// TIA Portal project "Apple_Juice_Process_System" (V15)
// Vorlageprojekt für das Buch mit Zielsystem S7-1200

(* hardware
DEVICE "S7-1200-Station_1"  S7-1200 Station
   slot 0: "Baugruppenträger_0"  Rack  V1.0
   slot 1: "PLC_1"  CPU 1211C DC/DC/DC  6ES7 211-1AE40-0XB0  V4.1
*)

// ===== PLC "PLC_1"  CPU 1211C DC/DC/DC =====

VAR_GLOBAL   // PLC tag table "Standard-Variablentabelle"
   "Tag_1" AT %Q1.6 : Bool;
   "Tag_2" AT %I1.5 : Bool;
   "Tag_3" AT %I1.6 : Bool;
   "System_Byte" AT %MB1 : Byte;
   "FirstScan" AT %M1.0 : Bool;
   "DiagStatusUpdate" AT %M1.1 : Bool;
   "AlwaysTRUE" AT %M1.2 : Bool;
   "AlwaysFALSE" AT %M1.3 : Bool;
   "Clock_Byte" AT %MB0 : Byte;
   "Clock_10Hz" AT %M0.0 : Bool;
   "Clock_5Hz" AT %M0.1 : Bool;
   "Clock_2.5Hz" AT %M0.2 : Bool;
   "Clock_2Hz" AT %M0.3 : Bool;
   "Clock_1.25Hz" AT %M0.4 : Bool;
   "Clock_1Hz" AT %M0.5 : Bool;
   "Clock_0.625Hz" AT %M0.6 : Bool;
   "Clock_0.5Hz" AT %M0.7 : Bool;
END_VAR

VAR_GLOBAL   // PLC tag table "I/O"
   "EMERGENCY_BUTTON" AT %I0.0 : Bool;
   "START_BUTTON" AT %I0.1 : Bool;
   "STOP_BUTTON" AT %I0.2 : Bool;
   "WATER_FLOW_METER" AT %ID30 : DWord;
   "WATER_LEVEL_METER" AT %ID34 : DWord;
   "APPLE_JUICE_FLOW_METER" AT %ID38 : DWord;
   "APPLE_JUICE_LEVEL_METER" AT %ID42 : DWord;
   "APPLE_FLOW_METER" AT %ID46 : DWord;
   "APPLE_LEVEL_METER" AT %ID50 : DWord;
   "ROLLER_ENABLE_0" AT %Q0.7 : Bool;
   "START_BUTTON_LIGHT" AT %Q0.1 : Bool;
   "STOP_BUTTON_LIGHT" AT %Q0.2 : Bool;
   "RESET_BUTTON_LIGHT" AT %Q0.3 : Bool;
   "WATER_CHARGE_VALVE" AT %QD30 : DWord;
   "WATER_DISCHARGE_VALVE" AT %QD34 : DWord;
   "APPLE_JUICE_CHARGE_VALVE" AT %QD38 : DWord;
   "APPLE_JUICE_DISCHARGE_VALVE" AT %QD42 : DWord;
   "APPLE_CHARGE_VALVE" AT %QD46 : DWord;
   "APPLE_DISCHARGE_VALVE" AT %QD50 : DWord;
   "PRODUCTION_ENABLE" AT %I0.3 : Bool;
   "PRODUCTION_DISABLE" AT %I0.4 : Bool;
   "APPLE_JUICE_AMOUNT_SET" AT %ID54 : DWord;
   "GREEN_LIGHT" AT %Q0.4 : Bool;
   "YELLOW_LIGHT" AT %Q0.5 : Bool;
   "RED_LIGHT" AT %Q0.6 : Bool;
   "HMI" AT %QD54 : DWord;
   "BOTTLE_LEFT" AT %I0.5 : Bool;
   "RESET_BUTTON" AT %I0.6 : Bool;
   "ROLLER_ENABLE_1" AT %Q1.0 : Bool;
   "ROLLER_ENABLE_2" AT %Q1.1 : Bool;
   "ROLLER_ENABLE_3" AT %Q1.2 : Bool;
END_VAR

DATA_BLOCK "main_prog_DB"   // DB1
{ S7_Optimized_Access := 'TRUE' }
VERSION : 0.1
// stored: InstanceOfName main_prog
"main_prog"
BEGIN
END_DATA_BLOCK

// folder: System blocks/Program resources

DATA_BLOCK "IEC_Timer_0_DB"   // DB7
{ S7_Optimized_Access := 'TRUE' }
AUTHOR : Simatic
FAMILY : IEC
NAME : IEC_TMR
VERSION : 1.0
// stored: InstanceOfName IEC_TIMER
"IEC_TIMER"
BEGIN
END_DATA_BLOCK

// folder: (top level)

FUNCTION_BLOCK "main_prog"   // FB1, SCL
{ S7_Optimized_Access := 'TRUE' }
VERSION : 0.1
   VAR_INPUT
      emergencyButton : Bool;
      startButton : Bool;
      stopButton : Bool;
      resetButton : Bool;
      productionEnable : Bool;
      productionDisable : Bool;
      bottleLeft : Bool;
      waterFlowMeter : Real;
      waterLevelMeter : Real;
      appleJuiceFlowMeter : Real;
      appleJuiceLevelMeter : Real;
      appleFlowMeter : Real;
      appleLevelMeter : Real;
      appleJuiceAmountSet : Real;
   END_VAR
   VAR_OUTPUT
      rollerEnable0 : Bool;
      rollerEnable1 : Bool;
      rollerEnable2 : Bool;
      rollerEnable3 : Bool;
      startButtonLight : Bool;
      stopButtonLight : Bool;
      resetButtonLight : Bool;
      greenLight : Bool;
      yellowLight : Bool;
      redLight : Bool;
      waterChargeValve : Real;
      waterDischargeValve : Real;
      appleJuiceChargeValve : Real;
      appleJuiceDischargeValve : Real;
      appleChargeValve : Real;
      appleDischargeValve : Real;
      hmi : Real;
   END_VAR
   VAR
      currentState : Int;
      risingEgdeDedect : Bool;
      fallingEgdeDedect : Bool;
      emergencyFallingEgdeDedect : Bool;
      stopButtonFallingEgdeDedect : Bool;
      stopRequested : Bool;
      requestedJuiceL : Real;
      appleTankChraged : Bool;
      waterTankChraged : Bool;
      appleTankDischarged : Bool;
      appleJuiceTankDischarged : Bool;
      waterTankDischarged : Bool;
      waterNeededForJuice : Real;
      appleNeededForJuice : Real;
      appleTankValue : Real;
      waterTankValue : Real;
      appleJuiceValue : Real;
      appleDischargeValue : Real;
      waterDischargeValue : Real;
      bottleValue : Real;
      emergencyState : Bool;
      bottleCounter : Real;
      savedState : Int;
      "timer" : Time;
      onDelayCheck : Bool;
      waitTime : Time := T#2s;
   END_VAR
   VAR CONSTANT
      STATE_INIT : Int;
      STATE_WAIT_FOR_START_AND_SAVE_APPLE_JUICE_VALUE : Int := 1;
      STATE_FILL_APPLE_AND_WATER_TANK : Int := 2;
      STATE_WAIT_FOR_FILL_UP : Int := 3;
      STATE_CALCULATE_JUICE_CONSTANTS : Int := 4;
      STATE_START_FILL_APPLE_JUICE_TANK_WITH_APPLE : Int := 5;
      STATE_WAIT_APLE_JUICE_FILL_UP_APPLE : Int := 6;
      STATE_START_FILL_APPLE_JUICE_TANK_WITH_WATER : Int := 7;
      STATE_WAIT_APLE_JUICE_FILL_UP_WATER : Int := 8;
      STATE_CALCULATE_BOTTLE_VALUE : Int := 9;
      STATE_START_FILL_BOTTLE : Int := 10;
      STATE_WAIT_FILL_BOTTLE : Int := 11;
      STATE_START_BOTTLE_CONVEYER : Int := 12;
      STATE_STOP_BOTTLE_CONVEYER : Int := 13;
      STATE_CHECK_FOR_WATER_AND_APPLE : Int := 14;
      STATE_START_DRAIN_ALL_TANKS : Int := 15;
      STATE_WAIT_DRAIN_ALL_TANKS : Int := 16;
      STATE_LIGHT_UP_RED_LIGHT : Int := 17;
      MAX_CHARGE : Real := 10.0;
      MAX_CHARGE_LEVEL : Real := 9.5;
      DISABLE_CHARGE : Real;
      DISABLE_DISCHARGE : Real;
      CLEAR_DISPLAY : Real;
      APPLE_PRECENT : Real := 70.0;
      WATER_PRECENT : Real := 30.0;
      TANK_DISCHARGE_VALUE : Real := 0.1;
      MINIMUM_BOTTLE_VALUE_IN_L : Real := 1.0;
   END_VAR
BEGIN
   "F_TRIG_DB_1"(CLK:=#emergencyButton,
                 Q=>#emergencyFallingEgdeDedect);

   "F_TRIG_DB_2"(CLK:=#stopButton,
                 Q=>#stopButtonFallingEgdeDedect);

   IF #stopButtonFallingEgdeDedect THEN
       #stopRequested := TRUE;
       #stopButtonLight := TRUE;
   END_IF;

   IF #emergencyFallingEgdeDedect THEN
       #emergencyState := TRUE;
       #savedState := #currentState;
       #currentState := -1;
   END_IF;

   IF #emergencyState THEN
       #waterChargeValve := #DISABLE_CHARGE;
       #waterDischargeValve := #DISABLE_DISCHARGE;

       #appleJuiceChargeValve := #DISABLE_CHARGE;
       #appleJuiceDischargeValve := #DISABLE_DISCHARGE;

       #appleChargeValve := #DISABLE_CHARGE;
       #appleDischargeValve := #DISABLE_DISCHARGE;

       #rollerEnable0 := FALSE;

       #startButtonLight := FALSE;
       #stopButtonLight := FALSE;
       #resetButtonLight := TRUE;

       #greenLight := FALSE;
       #yellowLight := FALSE;

       #redLight := "Clock_0.5Hz";

       "R_TRIG_DB_1"(CLK := #resetButton,
                     Q => #risingEgdeDedect);

       IF #risingEgdeDedect = TRUE AND #emergencyButton = TRUE THEN
           #emergencyState := FALSE;
           #redLight := FALSE;
           #resetButtonLight := FALSE;

           CASE #savedState OF
               #STATE_WAIT_FOR_FILL_UP:
                   #currentState := #STATE_FILL_APPLE_AND_WATER_TANK;

               #STATE_WAIT_APLE_JUICE_FILL_UP_APPLE:
                   #currentState := #STATE_START_FILL_APPLE_JUICE_TANK_WITH_APPLE;

               #STATE_WAIT_APLE_JUICE_FILL_UP_WATER:
                   #currentState := #STATE_START_FILL_APPLE_JUICE_TANK_WITH_WATER;

               #STATE_WAIT_FILL_BOTTLE:
                   #currentState := #STATE_START_FILL_BOTTLE;

               #STATE_STOP_BOTTLE_CONVEYER:
                   #currentState := #STATE_START_BOTTLE_CONVEYER;
               ELSE
                   #currentState := #savedState;
           END_CASE;
       END_IF;
   END_IF;

   CASE #currentState OF
       #STATE_INIT:
           #waterChargeValve := #DISABLE_CHARGE;
           #waterDischargeValve := #DISABLE_DISCHARGE;

           #appleJuiceChargeValve := #DISABLE_CHARGE;
           #appleJuiceDischargeValve := #DISABLE_DISCHARGE;

           #appleChargeValve := #DISABLE_CHARGE;
           #appleDischargeValve := #DISABLE_DISCHARGE;

           #stopButtonLight := FALSE;
           #startButtonLight := FALSE;
           #resetButtonLight := FALSE;

           #greenLight := FALSE;
           #yellowLight := FALSE;
           #greenLight := FALSE;

           #currentState := #STATE_WAIT_FOR_START_AND_SAVE_APPLE_JUICE_VALUE;

       #STATE_CHECK_FOR_WATER_AND_APPLE:
           #waterNeededForJuice := (#requestedJuiceL * #WATER_PRECENT) / 100.0;
           #appleNeededForJuice := (#requestedJuiceL * #APPLE_PRECENT) / 100.0;

           IF (#appleLevelMeter >= #appleNeededForJuice) AND
               (#waterLevelMeter >= #waterNeededForJuice) THEN

               #waterTankValue := #waterLevelMeter;
               #appleTankValue := #appleLevelMeter;

               #currentState := #STATE_CALCULATE_JUICE_CONSTANTS;
           ELSE
               #waterTankChraged := FALSE;
               #appleTankChraged := FALSE;

               #currentState := #STATE_FILL_APPLE_AND_WATER_TANK;
           END_IF;

       #STATE_WAIT_FOR_START_AND_SAVE_APPLE_JUICE_VALUE:
           #hmi := #appleJuiceAmountSet;
           #stopButtonLight := #productionDisable;
           #startButtonLight := #productionEnable;
           #yellowLight := TRUE;
           #greenLight := FALSE;
           #redLight := FALSE;

           "R_TRIG_DB"(CLK := #startButton,
                       Q => #risingEgdeDedect);

           IF #risingEgdeDedect THEN
               IF #productionEnable AND (#appleJuiceAmountSet > 0.0) THEN
                   #requestedJuiceL := #appleJuiceAmountSet;
                   #hmi := #CLEAR_DISPLAY;
                   #yellowLight := "Clock_5Hz";

                   #waterTankChraged := FALSE;
                   #appleTankChraged := FALSE;

                   #currentState := #STATE_FILL_APPLE_AND_WATER_TANK;

               ELSE
                   #currentState := #STATE_LIGHT_UP_RED_LIGHT;
               END_IF;
           END_IF;

           #STATE_LIGHT_UP_RED_LIGHT:
               "IEC_Timer_0_DB".TON(IN:=TRUE,
                                    PT:= #waitTime,
                                    ET => #timer,
                                    Q => #onDelayCheck);

               #redLight := TRUE;
               #yellowLight := FALSE;


               IF #onDelayCheck = TRUE THEN
                   "IEC_Timer_0_DB".TON(IN := FALSE,
                                        PT := #waitTime);
                   #redLight := FALSE;
                   #currentState := #STATE_WAIT_FOR_START_AND_SAVE_APPLE_JUICE_VALUE;
               END_IF;

       #STATE_FILL_APPLE_AND_WATER_TANK:
           #yellowLight := FALSE;
           #greenLight := TRUE;

           #waterChargeValve := #MAX_CHARGE;
           #appleChargeValve := #MAX_CHARGE;

           #currentState := #STATE_WAIT_FOR_FILL_UP;

       #STATE_WAIT_FOR_FILL_UP:
           IF #waterLevelMeter >= #MAX_CHARGE_LEVEL THEN
               #waterChargeValve := 0;
               #waterTankValue := #waterLevelMeter;
               #waterTankChraged := TRUE;
           END_IF;

           IF #appleLevelMeter >= #MAX_CHARGE_LEVEL THEN
               #appleChargeValve := 0;
               #appleTankValue := #appleLevelMeter;
               #appleTankChraged := TRUE;
           END_IF;

           IF #waterTankChraged = TRUE AND #appleTankChraged = TRUE THEN
               #currentState := #STATE_CALCULATE_JUICE_CONSTANTS;
           END_IF;

       #STATE_CALCULATE_JUICE_CONSTANTS:
           #waterTankValue := #waterLevelMeter;
           #appleTankValue := #appleLevelMeter;

           #waterNeededForJuice := (#requestedJuiceL * #WATER_PRECENT) / 100.0;
           #appleNeededForJuice := (#requestedJuiceL * #APPLE_PRECENT) / 100.0;

           #waterDischargeValue := #waterTankValue - #waterNeededForJuice;
           #appleDischargeValue := #appleTankValue - #appleNeededForJuice;

           #currentState := #STATE_START_FILL_APPLE_JUICE_TANK_WITH_APPLE;

       #STATE_START_FILL_APPLE_JUICE_TANK_WITH_APPLE:
           #appleDischargeValve := #MAX_CHARGE;
           #appleJuiceChargeValve := #MAX_CHARGE;

           #currentState := #STATE_WAIT_APLE_JUICE_FILL_UP_APPLE;

       #STATE_WAIT_APLE_JUICE_FILL_UP_APPLE:
           IF #appleLevelMeter <=  #appleDischargeValue THEN
               #appleDischargeValve := #DISABLE_DISCHARGE;
               #appleJuiceChargeValve := #DISABLE_CHARGE;

               #currentState := #STATE_START_FILL_APPLE_JUICE_TANK_WITH_WATER;
           END_IF;

       #STATE_START_FILL_APPLE_JUICE_TANK_WITH_WATER:
           #waterDischargeValve := #MAX_CHARGE;
           #appleJuiceChargeValve := #MAX_CHARGE;

           #currentState := #STATE_WAIT_APLE_JUICE_FILL_UP_WATER;

       #STATE_WAIT_APLE_JUICE_FILL_UP_WATER:
           IF #waterLevelMeter <= #waterDischargeValue THEN
               #waterDischargeValve := #DISABLE_DISCHARGE;
               #appleJuiceChargeValve := #DISABLE_CHARGE;
               #appleJuiceValue := #appleJuiceLevelMeter;

               #currentState := #STATE_CALCULATE_BOTTLE_VALUE;
           END_IF;

       #STATE_CALCULATE_BOTTLE_VALUE:
           #appleJuiceValue := #appleJuiceLevelMeter;
           #bottleValue := #appleJuiceValue - 1.0;

           IF #bottleValue >= #MINIMUM_BOTTLE_VALUE_IN_L THEN
               #currentState := #STATE_START_BOTTLE_CONVEYER;
           ELSE
               IF #stopRequested THEN
                   #stopRequested := FALSE;
                   #currentState := #STATE_START_DRAIN_ALL_TANKS;
                   #redLight := TRUE;
                   #greenLight := FALSE;
               ELSE
                   #currentState := #STATE_CHECK_FOR_WATER_AND_APPLE;
               END_IF;
           END_IF;

       #STATE_START_BOTTLE_CONVEYER:
           #rollerEnable0 := TRUE;
           #rollerEnable1 := TRUE;
           #rollerEnable2 := TRUE;
           #rollerEnable3 := TRUE;

           #currentState := #STATE_STOP_BOTTLE_CONVEYER;

       #STATE_STOP_BOTTLE_CONVEYER:
           "R_TRIG_DB_3"(CLK:=#bottleLeft,
                         Q=>#risingEgdeDedect);


           IF #risingEgdeDedect THEN
               #bottleCounter += 1;
               #hmi := #bottleCounter;

               #rollerEnable0 := FALSE;
               #rollerEnable1 := FALSE;
               #rollerEnable2 := FALSE;
               #rollerEnable3 := FALSE;
               #currentState := #STATE_START_FILL_BOTTLE; 
           END_IF;


       #STATE_START_FILL_BOTTLE:
           #appleJuiceDischargeValve := #MAX_CHARGE;

           #currentState := #STATE_WAIT_FILL_BOTTLE;

       #STATE_WAIT_FILL_BOTTLE:
           IF #appleJuiceLevelMeter <= #bottleValue THEN
               #appleJuiceDischargeValve := #DISABLE_DISCHARGE;

               #currentState := #STATE_CALCULATE_BOTTLE_VALUE;
           END_IF;

       #STATE_START_DRAIN_ALL_TANKS:
           #bottleCounter := 0;
           #hmi := #bottleCounter;

           #waterChargeValve := #DISABLE_CHARGE;
           #appleChargeValve := #DISABLE_CHARGE;
           #appleJuiceChargeValve := #DISABLE_CHARGE;

           #waterDischargeValve := #MAX_CHARGE;
           #appleDischargeValve := #MAX_CHARGE;
           #appleJuiceDischargeValve := #MAX_CHARGE;

           #waterTankDischarged := FALSE;
           #appleTankDischarged := FALSE;
           #appleJuiceTankDischarged := FALSE;

           #rollerEnable0 := FALSE;

           #currentState := #STATE_WAIT_DRAIN_ALL_TANKS;

       #STATE_WAIT_DRAIN_ALL_TANKS:
           IF #waterLevelMeter <= #TANK_DISCHARGE_VALUE THEN
               #waterDischargeValve := #DISABLE_DISCHARGE;
               #waterTankDischarged := TRUE;
           END_IF;

           IF #appleLevelMeter <= #TANK_DISCHARGE_VALUE THEN
               #appleDischargeValve := #DISABLE_DISCHARGE;
               #appleTankDischarged := TRUE;
           END_IF;

           IF #appleJuiceLevelMeter <= #TANK_DISCHARGE_VALUE THEN
               #appleJuiceDischargeValve := #DISABLE_DISCHARGE;
               #appleJuiceTankDischarged := TRUE;
           END_IF;

           IF #waterTankDischarged = TRUE
               AND #appleTankDischarged = TRUE
               AND #appleJuiceTankDischarged = TRUE THEN

               #waterDischargeValve := #DISABLE_DISCHARGE;
               #appleDischargeValve := #DISABLE_DISCHARGE;
               #appleJuiceDischargeValve := #DISABLE_DISCHARGE;

               #waterTankChraged := FALSE;
               #appleTankChraged := FALSE;

               #stopRequested := FALSE;

               #stopButtonLight := FALSE;

               #currentState := #STATE_WAIT_FOR_START_AND_SAVE_APPLE_JUICE_VALUE;
           END_IF;
   END_CASE;
END_FUNCTION_BLOCK

FUNCTION "MHJ-PLC-Lab-Function-S71200" : Void   // FC9000, SCL
{ S7_Optimized_Access := 'TRUE' }
VERSION : 0.1
   VAR_TEMP
      rdTimeReturn : Int;
      outputTime : DTL;
      SyncVal : Byte;
      forVal : Int;
      forVal_2 : Int;
      Value : Byte;
   END_VAR
   VAR CONSTANT
      CompVal : Byte := 16#34;
      Value_01 : Byte := 16#11;
      Value_01_DW : DWord := 16#A165_D992;
      Value_02_DW : DWord := 16#58BE_4401;
   END_VAR
BEGIN

   #Value:=PEEK(area := 16#82,
        dbNumber := 0,
        byteOffset := 511);
   #Value := #Value + 1;

   POKE(area := 16#82,
        dbNumber := 0,
        byteOffset := 511,
        value := #Value);

   POKE(area:=16#81,
        dbNumber:=0,
        byteOffset:=1016,
        value:=#Value_01_DW);
   POKE(area := 16#81,
        dbNumber := 0,
        byteOffset := 1020,
        value := #Value_02_DW);

   POKE(area := 16#81,
        dbNumber := 0,
        byteOffset := 511,
        value := B#16#00);

   FOR #forVal := 0 TO 120 DO
       FOR #forVal_2:=0 TO 10 DO
           #rdTimeReturn:=RD_SYS_T(#outputTime);
           #rdTimeReturn := WR_SYS_T(#outputTime);
           #rdTimeReturn := RD_SYS_T(#outputTime);
           #rdTimeReturn := WR_SYS_T(#outputTime);
       END_FOR;
       #SyncVal:= PEEK(area := 16#81,
                      dbNumber := 0,
                      byteOffset := 511);
       IF #SyncVal = #CompVal THEN
          GOTO M_1;
       END_IF;
   END_FOR;
   RETURN;

   M_1:
   POKE(area := 16#81,
        dbNumber := 0,
        byteOffset := 511,
        value := B#16#0);
END_FUNCTION

ORGANIZATION_BLOCK "Main"   // OB1, FBD, ProgramCycle
TITLE = "Main Program Sweep (Cycle)"
{ S7_Optimized_Access := 'TRUE' }
VERSION : 0.1
   VAR_INPUT
      Initial_Call : Bool;   // Initial call of this OB
      Remanence : Bool;   // =True, if remanent data are available
   END_VAR
BEGIN

REGION Network 1: Konnektierungsbaustein für PLC-Lab
   // Im Netzwerk 1 wird der Konnektierungsbaustein für PLC-Lab aufgerufen.
   // Dieser Aufruf darf nicht entfernt werden!
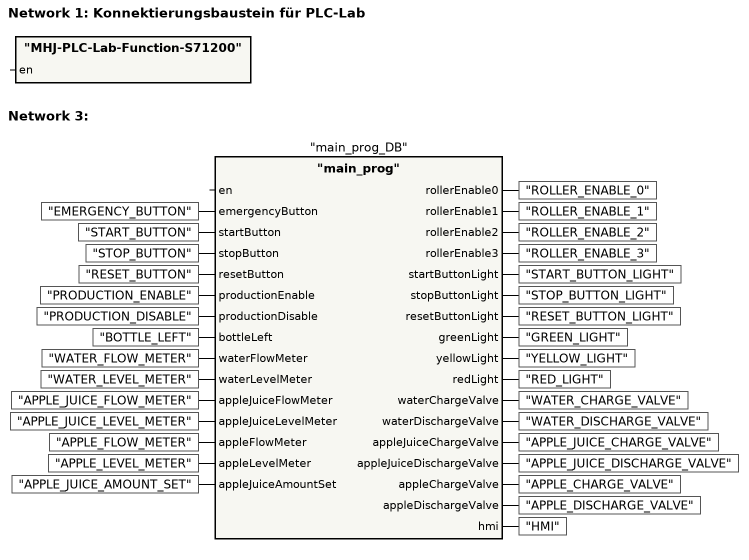
   "MHJ-PLC-Lab-Function-S71200"();
END_REGION

REGION Network 2: Ihr Programm
   // Schreiben Sie ab Netzwerk 2 Ihr Programm
END_REGION

REGION Network 3
   "main_prog_DB"(emergencyButton := "EMERGENCY_BUTTON",   // "main_prog"
                  startButton := "START_BUTTON",
                  stopButton := "STOP_BUTTON",
                  resetButton := "RESET_BUTTON",
                  productionEnable := "PRODUCTION_ENABLE",
                  productionDisable := "PRODUCTION_DISABLE",
                  bottleLeft := "BOTTLE_LEFT",
                  waterFlowMeter := "WATER_FLOW_METER",
                  waterLevelMeter := "WATER_LEVEL_METER",
                  appleJuiceFlowMeter := "APPLE_JUICE_FLOW_METER",
                  appleJuiceLevelMeter := "APPLE_JUICE_LEVEL_METER",
                  appleFlowMeter := "APPLE_FLOW_METER",
                  appleLevelMeter := "APPLE_LEVEL_METER",
                  appleJuiceAmountSet := "APPLE_JUICE_AMOUNT_SET",
                  rollerEnable0 => "ROLLER_ENABLE_0",
                  rollerEnable1 => "ROLLER_ENABLE_1",
                  rollerEnable2 => "ROLLER_ENABLE_2",
                  rollerEnable3 => "ROLLER_ENABLE_3",
                  startButtonLight => "START_BUTTON_LIGHT",
                  stopButtonLight => "STOP_BUTTON_LIGHT",
                  resetButtonLight => "RESET_BUTTON_LIGHT",
                  greenLight => "GREEN_LIGHT",
                  yellowLight => "YELLOW_LIGHT",
                  redLight => "RED_LIGHT",
                  waterChargeValve => "WATER_CHARGE_VALVE",
                  waterDischargeValve => "WATER_DISCHARGE_VALVE",
                  appleJuiceChargeValve => "APPLE_JUICE_CHARGE_VALVE",
                  appleJuiceDischargeValve => "APPLE_JUICE_DISCHARGE_VALVE",
                  appleChargeValve => "APPLE_CHARGE_VALVE",
                  appleDischargeValve => "APPLE_DISCHARGE_VALVE",
                  hmi => "HMI");
END_REGION
END_ORGANIZATION_BLOCK